TYPE LREAL_UNION :
UNION
    Value : LREAL;
    Raw : ULINT;
END_UNION
END_TYPE

(* stored: Version 1.1.0.1
   DUT LREAL_UNION: Id {0ec34dde-090d-4f4c-9891-07730a892d72} *)
